% RSLogix 500 project OR_PROJ_BAK009.RSS, saved by version 8.30.00.16 %
PROJECT "AND"    % processor: Bul.1763 MicroLogix 1100 Series B %

PROGRAM FILES
  LAD 2   2 rungs

DATA FILES
  O0 OUTPUT  4 elements
  I1 INPUT  6 elements
  S2 STATUS  66 elements
  B3 BINARY  1 elements
  T4 TIMER  1 elements
  C5 COUNTER  1 elements
  R6 CONTROL  1 elements
  N7 INTEGER  1 elements
  F8 FLOAT  1 elements

LADDER 2
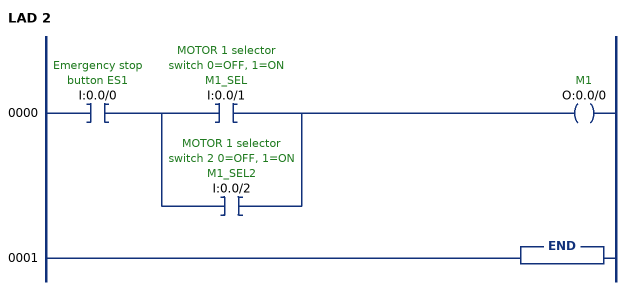
% Rung: 0 %
SOR XIC I:0.0/0 BST XIC I:0.0/1 NXB XIC I:0.0/2 BND OTE O:0.0/0 EOR
%   I:0.0/0  ES1  "Emergency stop button" %
%   I:0.0/1  M1_SEL  "MOTOR 1 selector switch 0=OFF, 1=ON" %
%   I:0.0/2  M1_SEL2  "MOTOR 1 selector switch 2 0=OFF, 1=ON" %
%   O:0.0/0  "M1" %
% Rung: 1 %
SOR END EOR

OTHER DOCUMENTED ADDRESSES
  B3:0/0  IN1
  B3:0/1  IN2
  B3:1/0  OU1
